// TwinCAT 3 PLC project Untitled1
// ProgramVersion: 3.1.4024.0
// libraries:
//   Tc2_Standard, * (Beckhoff Automation GmbH)
//   Tc2_System, * (Beckhoff Automation GmbH)
//   Tc3_Module, * (Beckhoff Automation GmbH)
//   VisuSymbols,3.5.10.0,System
// project tree:
//   / GlobalTextList.TcGTLO, PlcTask.TcTTO (not stored), PlcTask2.TcTTO (not stored), Visualization Manager.TcVMO (not stored)
//   GVLs/ GVL.TcGVL
//   POUs/ MAIN.TcPOU
//   VISUs/ Visualization.TcVIS
// real-time tasks:
//   TASK PlcTask: cycle T#10ms, priority 20, ADS port 350
//   TASK PlcTask2: cycle T#10ms, priority 21, ADS port 351

// ---- GVLs/GVL.TcGVL
{attribute 'qualified_only'}
VAR_GLOBAL
	Pressure_sensor : INT := 1;
	Pressure_Goal : INT := 1;
END_VAR

// ---- POUs/MAIN.TcPOU
PROGRAM MAIN
VAR
	Pressure_sensor : INT := 1;
	Pressure_Goal : INT := 1;	
	Pump_speed : INT := 0;
	Water_presence_sensor : BOOL;
	Water_presence_light : BOOL;
	
	Pump_on : BOOL;
	System_on : BOOL;
	System_off : BOOL;
	System_switch : BOOL;
END_VAR

IF system_switch THEN
	system_on := TRUE;
	system_off := FALSE;
ELSE
	system_on := FALSE;
	system_off := TRUE;
END_IF

IF Pressure_Goal < Pressure_sensor THEN
	IF Water_presence_sensor AND system_on THEN
		pump_on := TRUE;
	ELSE
		pump_on := FALSE;	
	END_IF
END_IF

IF water_presence_sensor THEN
	water_presence_light := TRUE;
ELSE
	water_presence_light := FALSE;
END_IF

IF Pump_on THEN
	IF Pump_speed < 100 THEN
		Pump_speed := Pump_speed + 1;
	END_IF
END_IF

IF NOT Pump_on THEN
	IF pump_speed > 1 THEN
		Pump_speed := Pump_speed - 1;
	END_IF
END_IF

END_PROGRAM

// ---- GlobalTextList.TcGTLO
TEXTLIST GlobalTextList
  510 = 'Button 1'
  435 = 'Drinking Beer'
  372 = 'Pressure goal'
  786 = 'Pressure sensor'
  376 = 'Pump'
  998 = 'Pump speed'
  276 = 'Sta vrij?'
  466 = 'System on/off'
  428 = 'Voetbal Training'
  282 = 'Water presence'
END_TEXTLIST

// ---- VISUs/Visualization.TcVIS
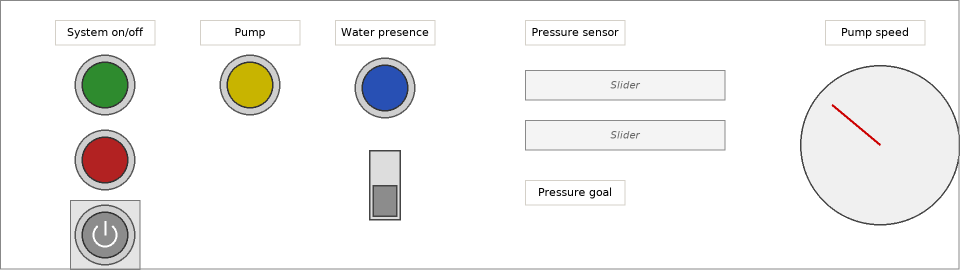
VISUALIZATION Visualization  // 960x270
    Lamp1 (70,50 70x70), variable: MAIN.System_on, style: Lamp-Lamp1-Green
    Slider (525,70 200x30), variable: MAIN.Pressure_sensor, scale 0..100
    PowerSwitch (70,200 70x70), variable: MAIN.System_switch, behaviour: TOGGLE, style: Switch-PowerSwitch-Gray
    Lamp1 (70,125 70x70), variable: MAIN.System_off, style: Lamp-Lamp1-Red
    Textfield (55,20 100x25), "System on/off"
    Textfield (200,20 100x25), "Pump"
    Lamp1 (215,50 70x70), variable: MAIN.Pump_on, style: Lamp-Lamp1-Yellow
    Lamp1 (350,53 70x70), variable: MAIN.Water_presence_light, style: Lamp-Lamp1-Blue
    Textfield (335,20 100x25), "Water presence"
    DipSwitch (350,150 70x70), variable: MAIN.Water_presence_sensor, behaviour: TOGGLE, style: Switch-DipSwitch-Gray
    Textfield (525,20 100x25), "Pressure sensor"
    Textfield (525,180 100x25), "Pressure goal"
    Slider (525,120 200x30), variable: MAIN.Pressure_Goal, scale 0..100
    Textfield (825,20 100x25), "Pump speed"
    Meter360 (800,65 160x160), value: MAIN.Pump_speed, style: Meter-Meter360-Gray, scale format: %.1f, scale 0..100
END_VISUALIZATION
